// Mitsubishi GX Works2 project: PLC 데이터 명령 (사칙연산)   PLC: Q03UDV

PROGRAM MAIN
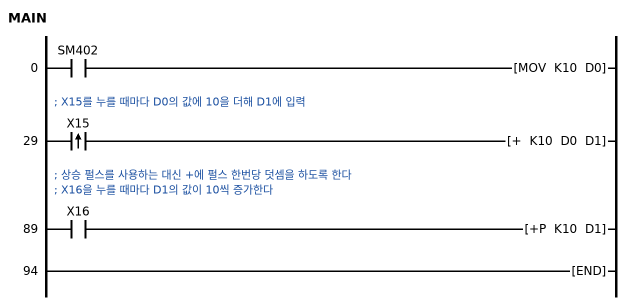
0     LD      SM402
      MOV     K10 D0
; X15를 누를 때마다 D0의 값에 10을 더해 D1에 입력
29    LDP     X15
      +       K10 D0 D1
; 상승 펄스를 사용하는 대신 +에 펄스 한번당 덧셈을 하도록 한다
; X16을 누를 때마다 D1의 값이 10씩 증가한다
89    LD      X16
      +P      K10 D1
94    END
END_PROGRAM
